// TIA Portal V20 export
// export: Created 2025-12-01T14:56:18.2075653Z, ExportSetting None, DisplayName Totally Integrated Automation Portal, DisplayVersion V20 Update 3, DisplayName TIA Portal Openness, DisplayVersion V20 Update 3, DisplayName TIA Portal Version Control Interface, DisplayVersion V20 Update 3, DisplayName STEP 7 Professional, DisplayVersion V20 Update 3, DisplayName STEP 7 Safety, DisplayVersion V20 Update 2, DisplayName WinCC Basic/Comfort/Advanced, DisplayVersion V20 Update 3, DisplayName WinCC Professional, DisplayVersion V20 Update 3, DisplayName WinCC Unified, DisplayVersion V20 Update 3
TYPE "VelMotor"
   STRUCT
      VelRapida_1 : Int;
      VelRapida_2 : Int;
      VelRapida_3 : Int;
      VelLenta_1 : Int;
      VelLenta_2 : Int;
      VelLenta_3 : Int;
      VelManual_1 : Int;
      VelManual_2 : Int;
      VelManual_3 : Int;
      Incremento_1 : Int;
      Incremento_2 : Int;
      Incremento_3 : Int;
   END_STRUCT;
END_TYPE
